(*

.. <legal notes>

legal notes
=================
| SPDX-FileCopyrightText: © 2026 Oleksandr Tiutyk <trofimich@gmail.com>
| SPDX-License-Identifier: LGPL-3.0-only
| For details check: LGPL-3.0-only_

.. _LGPL-3.0-only: https://www.gnu.org/licenses/lgpl-3.0.en.html

.. </legal notes>

*)

INTERFACE IIncompartibleGenericValueTypeException EXTENDS IGeneralException

END_INTERFACE

(* stored: Version 1.1.0.1
   Itf IIncompartibleGenericValueTypeException: Id {feeaa4aa-5b5e-462e-9c3e-1501eb3608c2} *)
